{attribute 'qualified_only'}
{attribute 'strict'}
TYPE E_MotorStates :
(
	stopped:=0,
	movingup,
	movingdown
);
END_TYPE

(* stored: Version 1.1.0.1, ProductVersion 3.1.4024.11
   DUT E_MotorStates: Id {55f9312d-4025-42a2-8830-49b8b58e865c} *)
